Fanuc TP program (LS listing): FOLGE125.LS

/PROG  FOLGE125
/ATTR
OWNER		= AUROM;
COMMENT		= "Pos. de Inicio";
PROG_SIZE	= 1136;
CREATE		= DATE 03-15-00  TIME 13:37:40;
MODIFIED	= DATE 17-02-24  TIME 03:42:10;
FILE_NAME	= ;
VERSION		= 0;
LINE_COUNT	= 6;
MEMORY_SIZE	= 2224;
PROTECT		= READ_WRITE;
TCD:  STACK_SIZE	= 500,
      TASK_PRIORITY	= 50,
      TIME_SLICE	= 0,
      BUSY_LAMP_OFF	= 0,
      ABORT_REQUEST	= 0,
      PAUSE_REQUEST	= 0;
DEFAULT_GROUP	= 1,1,1,1,*;
CONTROL_CODE	= 00000000 00000000;
/MN
   1:  UTOOL_NUM=1 ;
   2:  UFRAME_NUM=0 ;
   3:  PAYLOAD[1] ;
   4:J P[1] 10% CNT0 ACC100 TB   0.00sec,P-SPS    ;
      1:  IF (DO[12]=ON),CALL MAKRO998 ;
      2:  DO[15]=ON ;
      3:  DO[16]=ON ;
      4:  CALL MAKRO000    ;
      5:  WAIT (DI[9])    ;
       ------ ;
   5:  !Posicion de Inicio ;
   6:J P[2] 100% CNT0 ACC100 TB   0.00sec,P-SPS    ;
      1:  TC_ONLINE (ON) ;
      2:  DO[15]=OFF ;
      3:  DO[14]=ON ;
      4:  DO[15]=ON ;
       ------ ;
/POS
P[1]{
   GP1:
	UF : 0, UT : 1,
	J1=    90.000 deg,	J2=   -35.000 deg,	J3=    65.000 deg,
	J4=   180.000 deg,	J5=    80.000 deg,	J6=   -90.000 deg
   GP2:
	UF : 0, UT : 1,
	J1=   100.000  mm
   GP3:
	UF : 0, UT : 1,
	J1=     0.000  mm
   GP4:
	UF : 0, UT : 1,
	J1=     0.000  mm
};
P[2]{
   GP1:
	UF : 0, UT : 1,		CONFIG : 'F U T, 0, 1, 0',
	X =   317.190  mm,	Y =   894.706  mm,	Z =  2184.774  mm,
	W =     0.000 deg,	P =    15.000 deg,	R =    90.000 deg
   GP2:
	UF : 0, UT : 1,
	J1=   100.000  mm
   GP3:
	UF : 0, UT : 1,
	J1=     0.000  mm
   GP4:
	UF : 0, UT : 1,
	J1=     0.000  mm
};
/END
